INTERFACE ITF_BaseHMIGroupElement_View EXTENDS ITF_BaseHMIControlElement_View

END_INTERFACE

(* stored: Version 1.1.0.1
   Itf ITF_BaseHMIGroupElement_View: Id {21cd6ebf-8ae8-0215-3557-71ade5490935} *)
